VAR_GLOBAL CONSTANT
	nMaxTestSteps : UINT := 100;
END_VAR

VAR_GLOBAL
	nActiveTestStep	: UINT := 1;
	nActiveSubStep	: UINT := 0;
END_VAR

(* stored: Version 1.1.0.1
   GVL GVL_LeakTestConfig: Id {c83396cb-5407-08f9-090a-117fcfa39c5e} *)
